# EPICS substitutions: iocs/MC06/MCApp/Db-orig/SAI_GSCAN_Saver.substitutions
file /opt/epics/modules/genericScan/db/GSCAN_Saver.db {
pattern
{ 	P,		SCAN,		SCANREC,	FILESYSTEM,		SUBDIR}
	{ "FMB",	"GSCAN",	":SCANREC_SP",	"/opt/epics/iocoutput",	"gscandata" }
}
